FUNCTION_BLOCK HorizontalAct
VAR_INPUT
END_VAR
VAR_OUTPUT
	Extend		: BOOL;
	Extended	: BOOL;
	Retracted 	: BOOL;
	
END_VAR
VAR
END_VAR

METHOD mExtend : BOOL
VAR_INPUT
END_VAR
//IF ActInputs.Retracted AND Flags.PartReady THEN (Faulty)
//	Extend	:= ActOutputs.Extend := TRUE;
//END_IF
Extend	:= TRUE;
END_METHOD

METHOD mExtended : BOOL
VAR_INPUT
END_VAR
END_METHOD

METHOD mRetracted : BOOL
VAR_INPUT
END_VAR
END_METHOD

PROPERTY pExtend : BOOL
GET
pExtend	:= Extend;
END_GET
SET
Extend	:= pExtend;
END_SET
END_PROPERTY

PROPERTY pExtended : BOOL
GET
pExtended := Extended;
END_GET
SET
Extended := pExtended;
END_SET
END_PROPERTY

PROPERTY pRetracted : BOOL
GET
pRetracted := Retracted;
END_GET
SET
Retracted := pRetracted;
END_SET
END_PROPERTY

END_FUNCTION_BLOCK

(* stored: Version 1.1.0.1, ProductVersion 3.1.4024.9
   POU HorizontalAct: Id {0b4741e9-bb49-4cf0-9ec2-97a3053d9ff4}, SpecialFunc None
   Method mExtend: Id {edad9fd1-a486-4b17-8113-3f7c3c0cef09}
   Method mExtended: Id {c55d6d65-7b28-4ce8-80f8-40c35ce91e93}
   Method mRetracted: Id {53c2ff4a-4d34-4bcc-b668-7ff4667cb8d8}
   Property pExtend: Id {d477176f-dd99-4847-88f2-a8df32e10fc2}
   Get Get: Id {59cc3eac-02b1-48b9-9159-09d02d31d860}
   Set Set: Id {a6e1f594-83d0-48a3-b956-300fc67c3864}
   Property pExtended: Id {cd348aad-8aff-4110-848b-12151dcde4f6}
   Get Get: Id {804df2fd-f3ec-4260-86eb-0fa22e77ef87}
   Set Set: Id {8a972e77-8d5f-41b2-8a8d-c597841d73ee}
   Property pRetracted: Id {7d999191-23e5-4851-a4de-5efa3dcac5b1}
   Get Get: Id {bc3ba500-1bca-4bf2-88bf-e5cbc75505c4}
   Set Set: Id {797299eb-402d-4c6d-9663-d397f1cfb7bb} *)
